// TIA Portal V20 export
DATA_BLOCK "DB_GestionGripper"   // DB64
// stored: InstanceOfName FB_GestionGripper, InstanceOfType FB
"FB_GestionGripper"
   // VAR
   //    sLoadGripperCloseReq : Bool;
   //    sUnloadGripperCloseReq : Bool;
   //    sLoadShift : Bool;
   //    sUnLoadShift : Bool;
   //    sLoadPartLost : Bool;
   //    sUnLoadPartLost : Bool;
   //    sLoadClose : Bool;
   //    sUnLoadClose : Bool;
   //    sUndrilledGripper : "FB_Gripper";
   //    sDrilledGripper : "FB_Gripper";
   //    sLoadCloseWithPart : Bool;
   //    sUnLoadCloseWithPart : Bool;
   //    sLoadOpen : Bool;
   //    sUnLoadOpen : Bool;
   //    sFT_ModeJog : F_TRIG;
   //    sBlowingTimerCmdHMI : TP_TIME;
   //    sRT_BlowingCmdHMI { S7_SetPoint := 'True'} : R_TRIG;
   //    sBlowingISO { S7_SetPoint := 'True'} : Bool;
   //    sGripperStatus : Struct
   //       Available : Bool;
   //       DrivedByShuttle1 : Bool;
   //       DrivedByShuttle2 : Bool;
   //       DrivedByFixture : Bool;
   //    END_STRUCT;
   //    sGripperReq : Struct
   //       ByShuttle1 : Bool;
   //       ByShuttle2 : Bool;
   //       ByFixture : Bool;
   //    END_STRUCT;
   //    sUndrilledGripperErrorCode : Int;
   //    sDrilledGripperErrorCode : Int;
   // END_VAR
BEGIN
END_DATA_BLOCK
